(* PLC project batch, Dassault Systèmes ControlBuild 2024x *)
(* stored: creationDateTime 2023-10-05T15:42:43-01:00 *)

CONFIGURATION batch
  VAR_GLOBAL
    simuperiod : REAL := 50000.0;
    taskname : STRING(50) := 'batch.exe';
    allowpreconditions : BOOL := true;
    allowpostconditions : BOOL := true;
    generalPanel/emergencyStop/PBLogic : BOOL := false;
    manufacturing/flour/airArrival/inputFlow : REAL := 50.0;
    manufacturing/flour/airArrival/valve/openingTime : REAL := 0.5;
    manufacturing/flour/extractingValve/valve/openingTime : REAL := 0.5;
    manufacturing/flour/airExtraction/valve/openingTime : REAL := 0.5;
    manufacturing/flour/flourWeighing/capacity : REAL := 100.0;
    manufacturing/flour/flow/flowMax : REAL := 20000.0;
    manufacturing/syrup/flow/flowMax : REAL := 40000.0;
    manufacturing/syrup/arrivalValveSyrup1/inputFlow : REAL := 50.0;
    manufacturing/syrup/arrivalValveSyrup1/valve/openingTime : REAL := 0.5;
    manufacturing/syrup/arrivalValveSyrup2/inputFlow : REAL := 50.0;
    manufacturing/syrup/arrivalValveSyrup2/valve/openingTime : REAL := 0.5;
    manufacturing/syrup/arrivalValveSyrup3/inputFlow : REAL := 50.0;
    manufacturing/syrup/arrivalValveSyrup3/valve/openingTime : REAL := 0.5;
    manufacturing/syrup/syrupExtractionValve/valve/openingTime : REAL := 0.5;
    manufacturing/syrup/syrupsTank/capacity : REAL := 300.0;
    manufacturing/syrup/scale/maxInput : REAL := 300.0;
    manufacturing/syrup/scale/maxOutput : REAL := 300.0;
    manufacturing/mixture/flow/flowMax : REAL := 40000.0;
    manufacturing/mixture/mixtureWeighing/capacity : REAL := 600.0;
    manufacturing/mixture/scale/maxInput : REAL := 600.0;
    manufacturing/mixture/scale/maxOutput : REAL := 600.0;
  END_VAR
END_CONFIGURATION
